// TIA Portal V20 export
DATA_BLOCK "RealDbName"   // DB8
   VAR
      InternalCalcBuffer { ExternalAccessible := 'False'; ExternalVisible := 'False'; ExternalWritable := 'False'} : Array[0..9] of Real;
   END_VAR
BEGIN
END_DATA_BLOCK
